Staubli VAL3: GetKeyIO.pgx

public program GetKeyIO(bool& x_AirOn (dimensions=1), bool& x_bFollowOn (dimensions=1), bool& x_bLaserOn (dimensions=1))
  local string l_sS
begin

  //气体
  call IOName(70,l_sS)
  x_AirOn=dDio[l_sS]==true


  //随动
  call IOName(68,l_sS)
  x_bFollowOn=dDio[l_sS]==true


  //焊接
  if bWeldEnable
    call IOName(79,l_sS)
    x_bLaserOn=dDio[l_sS]==true

  else
    //   切割
    call IOName(67,l_sS)
    x_bLaserOn=dDio[l_sS]==true
  endIf

end
